// SIMATIC S7-200 SMART project (STEP 7-Micro/WIN SMART), CPU ST40

SYMBOL_TABLE Table 1
Start_SW         I0.0
OFF_SW           I0.1
CARS_COUNTER     C1
CAR_IN           I0.2
MEMORY           M0.0
CLOSED           Q0.2
OPEN             Q0.1
CAR_OUT          I0.3
END_SYMBOL_TABLE

ORGANIZATION_BLOCK MAIN:OB1
TITLE=Program Comments
BEGIN
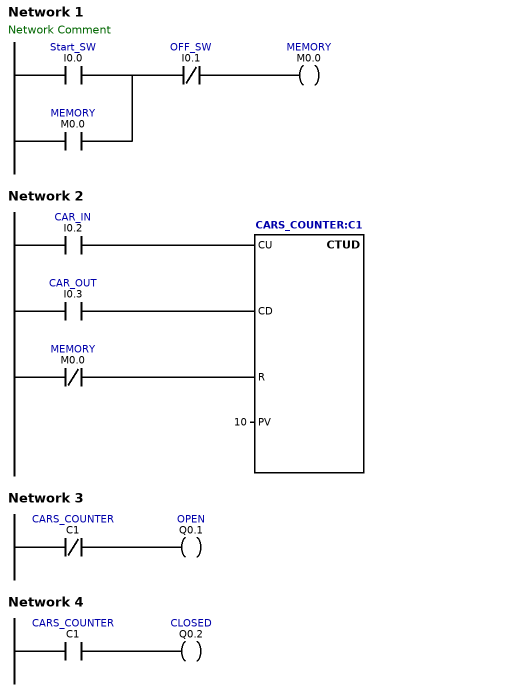
Network 1
// Network Comment
LD     Start_SW:I0.0
O      MEMORY:M0.0
AN     OFF_SW:I0.1
=      MEMORY:M0.0
Network 2
LD     CAR_IN:I0.2
LD     CAR_OUT:I0.3
LDN    MEMORY:M0.0
CTUD   CARS_COUNTER:C1, 10
Network 3
LDN    CARS_COUNTER:C1
=      OPEN:Q0.1
Network 4
LD     CARS_COUNTER:C1
=      CLOSED:Q0.2
END_ORGANIZATION_BLOCK
